// TIA Portal V19 export
DATA_BLOCK "AO SCALING DB"   // DB170
{ S7_Optimized_Access := 'FALSE' }
   VAR
      SET : Struct
         "VFD P-301A" : Real;
         "VFD P-301B" : Real;
         "VFD P-402A" : Real;
         "VFD P-402B" : Real;
      END_STRUCT;
      MIN : Struct
         "VFD P-301A" : Real;
         "VFD P-301B" : Real;
         "VFD P-402A" : Real;
         "VFD P-402B" : Real;
         "VFD P-501A_7" : Real;
      END_STRUCT;
      MAX : Struct
         "VFD P-301A" { S7_SetPoint := 'True'} : Real := 50.0;
         "VFD P-301B" { S7_SetPoint := 'True'} : Real := 50.0;
         "VFD P-402A" { S7_SetPoint := 'True'} : Real := 50.0;
         "VFD P-402B" { S7_SetPoint := 'True'} : Real := 50.0;
         "VFD P-501A_7" : Real;
      END_STRUCT;
      PV : Struct
         "VFD P-301A" : Int;
         "VFD P-301B" : Int;
         "VFD P-402A" : Int;
         "VFD P-402B" : Int;
      END_STRUCT;
   END_VAR
BEGIN
END_DATA_BLOCK
